TYPE DEBUG_SKILL :
STRUCT
	bExecute,bStop : BOOL;
END_STRUCT
END_TYPE

(* stored: Version 1.1.0.1, ProductVersion 3.1.4026.18
   DUT DEBUG_SKILL: Id {3ef44a0b-a33b-43ed-a1d4-8190adbd6929} *)
